// TIA Portal project "Tank valve PID" (V18)

(* hardware
DEVICE "S71500/ET200MP station_1"  S7-1500 station
   slot 0: "Rail_0"  Rack  6ES7 590-1***0-0AA0
   slot 1: "Controller"  CPU 1512C-1 PN  6ES7 512-1CK01-0AB0  V2.5
      slot 3: "CPU display_1"  6ES7591-1AA00-0AA0
DEVICE "System_View"  SIMATIC PC station
   slot 0: "SIMATIC PC station"  Rail  SIMATIC PC-Station  V1.0
      slot 125: "Stationmanager"  Station_Manager  V6.0.4
   slot 1: "HMI_RT_1"  WinCC RT Advanced  6AV2 104-0xxxx-xxxx  15.1.0.0
      slot 33792: "Host interface"  Host interface
   slot 2: "IE general_1"  IE General  IE_CP  V8.2.0
*)

// ===== PLC "Controller"  CPU 1512C-1 PN =====
// protected blocks, not shown: "Analog Input Processing", "Analog Output Processing", "Cyclic interrupt 1ms", "Main", "Manual Control", "ON/OFF Control", "ON/OFF Control w. Hysteresis", "Tank Behaviour FB"

VAR_GLOBAL   // PLC tag table "Default tag table"
   "Clock_Byte" AT %MB100 : Byte;
   "Clock_10Hz" AT %M100.0 : Bool;
   "Clock_5Hz" AT %M100.1 : Bool;
   "Clock_2.5Hz" AT %M100.2 : Bool;
   "Clock_2Hz" AT %M100.3 : Bool;
   "Clock_1.25Hz" AT %M100.4 : Bool;
   "Clock_1Hz" AT %M100.5 : Bool;
   "Clock_0.625Hz" AT %M100.6 : Bool;
   "Clock_0.5Hz" AT %M100.7 : Bool;
END_VAR

// folder: Data Bases

DATA_BLOCK "HMI Data"   // DB1
{ S7_Optimized_Access := 'TRUE' }
VERSION : 0.1
   VAR
      "Fill Level (in l)" : Real;
      "Setpoint (in l)" : Real;
      "Pump Flow (l/s)" : Real;   // Before Idle Time
      "PLC Output" : Int;
      "Disturbance (in %/s)" : Real := 5.0;
      "Manual Control (in %)" : Int;
      "Controller Type" : SInt;
      "Empty Tank" : Bool;
      "Tolerance (in l)" : Real;
      "Idle Time (ms)" : Int := 2500;
      "Random Error" : SInt;
   END_VAR
BEGIN
END_DATA_BLOCK

DATA_BLOCK "Analog Data"   // DB3
{ S7_Optimized_Access := 'TRUE' }
VERSION : 0.1
   VAR
      "Fill Level PLC Input" : Int;
      "Calc PID" : Real;
   END_VAR
BEGIN
END_DATA_BLOCK

// folder: (top level)

ORGANIZATION_BLOCK "Cyclic interrupt PID"   // OB31, LAD, CyclicInterrupt
{ S7_Optimized_Access := 'TRUE' }
VERSION : 0.1
   VAR_INPUT
      Initial_Call : Bool;   // Initial call of this OB
      Event_Count : Int;   // Events discarded
   END_VAR
   VAR_TEMP
      Calc : Real;
   END_VAR
BEGIN

REGION Network 1
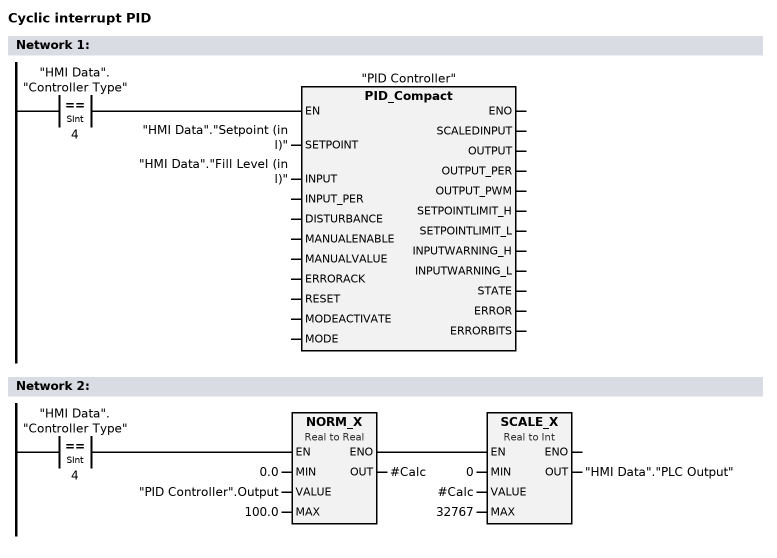
   IF "HMI Data"."Controller Type" = 4 THEN
       "PID Controller"(Setpoint := "HMI Data"."Setpoint (in l)", Input := "HMI Data"."Fill Level (in l)");   // PID_Compact
   END_IF;
END_REGION

REGION Network 2
   RUNG wire#powerrail
      { S7_Templates := "SrcType := SInt" } EQ_Contact(in1 := "HMI Data"."Controller Type", in2 := 4)
      { S7_Templates := "[SrcType := Real, DestType := Real]" } Normalize(min := 0.0, value := "PID Controller".Output, max := 100.0, out => #Calc)
      { S7_Templates := "[SrcType := Real, DestType := Int]" } Scale(min := 0, value := #Calc, max := 32767, out => "HMI Data"."PLC Output")
   END_RUNG
   // the same network as SCL:
   IF "HMI Data"."Controller Type" = 4 THEN
       #Calc := NORM_X(MIN := 0.0, VALUE := "PID Controller".Output, MAX := 100.0);
       "HMI Data"."PLC Output" := SCALE_X(MIN := 0, VALUE := #Calc, MAX := 32767);
   END_IF;
END_REGION
END_ORGANIZATION_BLOCK

(* ===== HMI "HMI_RT_1" =====
system functions are stored by id; their names below are inferred from use
connection "HMI_Connection_1": ETHERNET, S7_1500_OMS

HMI tags "Default tag table"
   "HMI Data_Fill Level" : Real = PLC "HMI Data"."Fill Level (in l)", 100 ms
   "HMI Data_Setpoint" : Real = PLC "HMI Data"."Setpoint (in l)", 100 ms
   "HMI Data_PLC Output" : Int = PLC "HMI Data"."PLC Output", 100 ms
   "HMI Data_Disturbance (%/s)" : Real = PLC "HMI Data"."Disturbance (in %/s)", 100 ms
   "HMI Data_Manual Control (%)" : Int = PLC "HMI Data"."Manual Control (in %)", 100 ms
   "HMI Data_Controller Type" : SInt = PLC "HMI Data"."Controller Type", 100 ms
   "HMI Data_Empty Tank" : Bool = PLC "HMI Data"."Empty Tank", 100 ms
   "HMI Data_Tolerance" : Real = PLC "HMI Data"."Tolerance (in l)", 100 ms
   "PID Controller_Retain_CtrlParams_Gain" : Real = PLC "PID Controller".Retain.CtrlParams.Gain, 100 ms
   "PID Controller_Retain_CtrlParams_Ti" : Real = PLC "PID Controller".Retain.CtrlParams.Ti, 100 ms
   "PID Controller_Retain_CtrlParams_Td" : Real = PLC "PID Controller".Retain.CtrlParams.Td, 100 ms
   "PID Controller_PIDCtrl_IntegralSum" : Real = PLC "PID Controller".PIDCtrl.IntegralSum, 100 ms
   "HMI Data_Idle Time" : Int = PLC "HMI Data"."Idle Time (ms)", 1 s
   "HMI Data_Random Error" : SInt = PLC "HMI Data"."Random Error", 1 s
   "PID Controller_Retain_CtrlParams_Cycle" : Real = PLC "PID Controller".Retain.CtrlParams.Cycle, 1 s

text list "Controller Type": 0 'OFF'; 2 'ON/OFF'; 3 'ON/OFF w. Hysteresis'; 4 'PID'; 1 'Manual'

text list "Random Error": 2 'Weak'; 3 'Medium'; 4 'Strong'; 1 'Off'; 0 'Off'

screen "Screen_1" 1024x768
   Bar "Bar_1" at 56,195 size 331x422; MinimumValue 0; MaximumValue 10
      ProcessValue <- "HMI Data_Fill Level"
   IOField "I/O field_1" at 169,94 size 108x32; FormatPattern 99.999; Unit  l
      ProcessValue <- "HMI Data_Setpoint"
      Visibility <- "HMI Data_Controller Type"
   TextField "Text field_1" at 56,99 size 112x22; Text 'Setpoint'
      Visibility <- "HMI Data_Controller Type"
   Slider "Slider_1" at 401,47 size 592x121; Caption 'Manual Control'
      ProcessValue <- "HMI Data_Manual Control (%)"
      Visibility <- "HMI Data_Controller Type"
   IOField "I/O field_2" at 228,629 size 160x32; FormatPattern 999.99; Unit  %/sec
      ProcessValue <- "HMI Data_Disturbance (%/s)"
   TextField "Text field_2" at 51,632 size 168x28; Text 'Outflow'
   TrendView "Trend view_1" at 401,198 size 592x479
   SymbolicIOField "Symbolic I/O field_1" at 56,45 size 220x32; TextOff '0'; TextOn '1'; TextList "Controller Type"
      ProcessValue <- "HMI Data_Controller Type"
   Button "Button_1" at 283,558 size 99x45; TextOff 'Empty Tank'
      on Press: function_b14e0dd5("HMI Data_Empty Tank", 0)
   IOField "I/O field_3" at 170,136 size 107x32; FormatPattern 9.999; Unit  l
      ProcessValue <- "HMI Data_Tolerance"
      Visibility <- "HMI Data_Controller Type"
   TextField "Text field_3" at 56,141 size 114x22; Text 'Tolerance'
      Visibility <- "HMI Data_Controller Type"
   IOField "I/O field_4" at 343,60 size 106x32
      ProcessValue <- "PID Controller_Retain_CtrlParams_Gain"
      Visibility <- "HMI Data_Controller Type"
   IOField "I/O field_5" at 343,97 size 106x32; Unit  s
      ProcessValue <- "PID Controller_Retain_CtrlParams_Ti"
      Visibility <- "HMI Data_Controller Type"
   IOField "I/O field_6" at 343,134 size 106x32; Unit  s
      ProcessValue <- "PID Controller_Retain_CtrlParams_Td"
      Visibility <- "HMI Data_Controller Type"
   TextField "Text field_4" at 463,67 size 187x22; Text 'Proportional Gain'
      Visibility <- "HMI Data_Controller Type"
   TextField "Text field_5" at 460,103 size 202x22; Text 'Ti - Reset Time'
      Visibility <- "HMI Data_Controller Type"
   TextField "Text field_6" at 462,140 size 190x22; Text 'Td - Derivative Time'
      Visibility <- "HMI Data_Controller Type"
   TextField "Text field_7" at 783,103 size 202x22; Text 'Integral Sum'
      Visibility <- "HMI Data_Controller Type"
   IOField "I/O field_7" at 650,97 size 121x32; FormatPattern 99999.999
      ProcessValue <- "PID Controller_PIDCtrl_IntegralSum"
      Visibility <- "HMI Data_Controller Type"
   TextField "Text field_10" at 23,676 size 197x28; Text 'Random Disturbance'
   SymbolicIOField "Symbolic I/O field_2" at 228,672 size 160x32; TextOff '0'; TextOn '1'; TextList "Random Error"
      ProcessValue <- "HMI Data_Random Error"
   IOField "EA-Feld_2" at 227,717 size 162x32; FormatPattern 9999; Unit  ms
      ProcessValue <- "HMI Data_Idle Time"
   TextField "Text field_8" at 25,717 size 197x28; Text 'Idle Time'
   IOField "I/O field_8" at 184,136 size 93x32; FormatPattern 9.999; Unit  s
      Visibility <- "HMI Data_Controller Type"
      ProcessValue <- "PID Controller_Retain_CtrlParams_Cycle"
   TextField "Text field_9" at 58,141 size 152x22; Text 'Sampling Time'
      Visibility <- "HMI Data_Controller Type"
*)